Yaskawa INFORM job: !TOOL-CHECK-BY-HAND!.JBI

/JOB
//NAME !TOOL-CHECK-BY-HAND!
//POS
///NPOS 17,17,0,0,0,0
///TOOL 0
///POSTYPE PULSE
///PULSE
C00000=0,0,-1,0,0,46844
C00001=12704,6043,-50274,122642,39769,-30984
C00002=12704,-8329,-23679,95263,52732,-11236
C00003=4271,-27562,-37322,97890,58327,-12168
C00004=-18291,-59373,-52766,85939,61827,-4486
C00005=1830,-5213,-26868,109844,57376,-17779
C00006=676,-4492,-28689,111788,57883,-20604
C00007=1830,-5213,-26868,109844,57376,-17779
C00008=2018,375,-22259,109354,57368,-17486
C00009=2140,772,-22694,110080,57052,-17963
C00010=2038,282,-22123,109103,57429,-17328
C00011=2038,282,-22123,109103,57429,-17328
C00012=2142,737,-22421,109744,57156,-17750
C00013=2038,282,-22123,109103,57429,-17328
C00014=12704,-8329,-23679,95263,52732,-11236
C00015=12704,6043,-50274,122642,39769,-30984
C00016=0,0,-1,0,0,46844
BC00000=175236
BC00001=106776
BC00002=106776
BC00003=106776
BC00004=106776
BC00005=106778
BC00006=106778
BC00007=106778
BC00008=106778
BC00009=106779
BC00010=106779
BC00011=106779
BC00012=106779
BC00013=106779
BC00014=106776
BC00015=106776
BC00016=175236
//INST
///DATE 2018/10/04 11:08
///ATTR SC,RW
///GROUP1 RB1,BS1
NOP
SFTOF
'"
'Checking tool on zero position
'"
*teach
MOVJ C00000 BC00000 VJ=25.00
'"
'Set register
SETREG MREG#(1) 1
'"
MOVL C00001 BC00001 V=166.7
'"
'Set register
SETREG MREG#(1) 3
'"
MOVL C00002 BC00002 V=166.7
'"
'Set register
SETREG MREG#(1) 4
'"
MOVL C00003 BC00003 V=166.7
'"
'Set register
SETREG MREG#(1) 4
'"
'********************************
'Maintenance pos
'"
MOVL C00004 BC00004 V=83.3 PL=0
PAUSE
'"
'Check position tool
'"
MOVL C00005 BC00005 V=166.7
MOVL C00006 BC00006 V=16.7 PL=0
'"
'"
'"
'Please check stick out
'"
'"
'"
MOVL C00007 BC00007 V=166.7
MOVL C00008 BC00008 V=166.7
MOVL C00009 BC00009 V=16.7 PL=0
PAUSE
'"
'"
'"
'Please check TCP off torch
'"
'"
'"
MOVL C00010 BC00010 V=166.7
MOVL C00011 BC00011 V=166.7
MOVL C00012 BC00012 V=16.7 PL=0
PAUSE
'"
'"
'"
'Please check TCP off wire
'"
'"
'"
'********************************
MOVL C00013 BC00013 V=166.7
'"
'"
MOVL C00014 BC00014 V=166.7
'"
'Set register
SETREG MREG#(1) 3
'"
MOVL C00015 BC00015 V=166.7
'"
'Set register
SETREG MREG#(1) 2
'"
MOVL C00016 BC00016 V=166.7
'"
'Set register
SETREG MREG#(1) 1
'"
END
